// Mitsubishi GX Works2 project: Prática 01 - L_D   PLC: FX3U/FX3UC
// Configuração Modbus RTU

PROGRAM MAIN
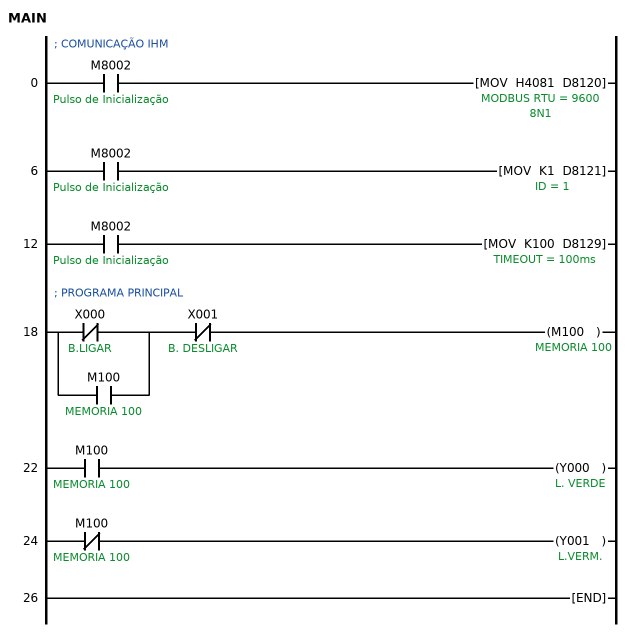
; COMUNICAÇÃO IHM
0     LD      M8002  ; Pulso de Inicialização
      MOV     H4081 D8120  ; MODBUS RTU = 9600 8N1
6     LD      M8002  ; Pulso de Inicialização
      MOV     K1 D8121  ; ID = 1
12    LD      M8002  ; Pulso de Inicialização
      MOV     K100 D8129  ; TIMEOUT = 100ms
; PROGRAMA PRINCIPAL
18    LDI     X000  ; B.LIGAR
      OR      M100  ; MEMORIA 100
      ANI     X001  ; B. DESLIGAR
      OUT     M100  ; MEMORIA 100
22    LD      M100  ; MEMORIA 100
      OUT     Y000  ; L. VERDE
24    LDI     M100  ; MEMORIA 100
      OUT     Y001  ; L.VERM.
26    END
END_PROGRAM

// device comments not shown above
Y002  ; RELE 2
Y004  ; MOTOR
Y005  ; SENTIDO
M0  ; VARIAVEL DE MEMORIA 0
M1  ; VARIAVEL DE MEMORIA 1
M2  ; VARIAVEL DE MEMORIA 2
D0  ; REGISTRO 0
D1  ; LEITURA 1
D2  ; ENCHE O TANQUE
D3  ; ESVAZIA O TANQUE
